// TIA Portal V20 export
TYPE "Log_Data_Char"
// stored: Namespace ProductionLine
   STRUCT
      DataType : Byte;
      Representation : Byte;
      RepreLength : Byte;
      Reserve : Byte;
      Data : Char;
   END_STRUCT;
END_TYPE
